FUNCTION F_Scale : REAL

VAR_INPUT
	inputValue : REAL;
	inputMaxValue : REAL;
	inputMinValue : REAL;
	inputScaleMaxLimit : REAL; 
	inputScaleMinLimit : REAL;
END_VAR

VAR
	fNormalizedValue : REAL :=0;
	fScaledValue : REAL := 0;
END_VAR

//Normalize the  input
IF inputValue < inputMinValue THEN
	fNormalizedValue := 0;
ELSIF inputValue > 	inputMaxValue THEN
	fNormalizedValue := 1;
ELSE
	fNormalizedValue := (inputValue - inputMinValue) / (inputMaxValue - inputMinValue);
END_IF

//Scale the output
F_Scale := fNormalizedValue * (inputScaleMaxLimit - inputScaleMinLimit) + inputScaleMinLimit;

END_FUNCTION

(* stored: Version 1.1.0.1, ProductVersion 3.1.4024.12
   POU F_Scale: Id {49775636-e960-4359-8a08-12d42221b5ac}, SpecialFunc None *)
